FUNCTION_BLOCK EM_Can_Supply IMPLEMENTS  ITF_EM_Can_Supply
VAR_INPUT
END_VAR
VAR_OUTPUT
END_VAR
VAR
END_VAR

END_FUNCTION_BLOCK

(* stored: Version 1.1.0.1, ProductVersion 3.1.4024.12
   POU EM_Can_Supply: Id {80e52e0b-6656-4ee1-942a-74f49012a38a}, SpecialFunc None *)
